{attribute 'linkalways'} 
{attribute 'no_explicit_call' := 'This FB is a CLASS and must be accessed using methods or properties'}
{attribute 'enable_dynamic_creation'}
FUNCTION_BLOCK _TcVnArray7_LREAL EXTENDS AliasDatatypeBase
VAR
	localData : TcVnArray7_LREAL;
	activeData : REFERENCE TO TcVnArray7_LREAL REF= localData;
	aliasBaseDatatype : _Array0to6OfLREAL;
END_VAR

PROPERTY PUBLIC Address : PVOID
GET
Address := ADR(activeData);
END_GET
END_PROPERTY

METHOD PUBLIC ClearReference
VAR_INPUT
END_VAR
activeData REF= localData;
SetBaseDatatypeReference();
END_METHOD

METHOD PUBLIC Clone : I_Datatype
VAR
    pClone : POINTER TO _TcVnArray7_LREAL;
END_VAR
pClone := __NEW(_TcVnArray7_LREAL);
Clone := pClone^;
END_METHOD

METHOD FB_init : BOOL
VAR_INPUT
	bInitRetains : BOOL; // if TRUE, the retain variables are initialized (warm start / cold start)
	bInCopyCode : BOOL;  // if TRUE, the instance afterwards gets moved into the copy code (online change)
	//InitialValue : TcVnArray7_LREAL; // if possible, not all values can be initialized
END_VAR
//localData := InitialValue; // if possible, not all values can be initialized
SetBaseDatatypeReference();
AddBaseDatatype(aliasBaseDatatype);
END_METHOD

PROPERTY PUBLIC Identifier : T_MAXSTRING
GET
Identifier := 'TcVnArray7_LREAL';
END_GET
END_PROPERTY

METHOD PUBLIC MakeReferenceTo
VAR_INPUT
	ReferenceTarget : REFERENCE TO TcVnArray7_LREAL;
END_VAR
activeData REF= ReferenceTarget;
SetBaseDatatypeReference();
END_METHOD

METHOD PROTECTED SetBaseDatatypeReference
VAR_INPUT
END_VAR
aliasBaseDatatype.MakeReferenceTo(activeData);
END_METHOD

PROPERTY PUBLIC Size : UDINT
GET
Size := SIZEOF(activeData);
END_GET
END_PROPERTY

METHOD TryMakeReferenceTo : BOOL
VAR_INPUT
	Target : I_Datatype;
END_VAR
VAR
	pTargetData : POINTER TO TcVnArray7_LREAL;
END_VAR
IF NOT IsEquivalentTo(Target) THEN
	RETURN;
END_IF

pTargetData := Target.Address;
activeData REF= pTargetData^;
SetBaseDatatypeReference();
TryMakeReferenceTo := TRUE;
END_METHOD

PROPERTY PUBLIC Value : REFERENCE TO TcVnArray7_LREAL
GET
Value REF= activeData;
END_GET
END_PROPERTY

END_FUNCTION_BLOCK

(* stored: Version 1.1.0.1, ProductVersion 3.1.4024.13
   POU _TcVnArray7_LREAL: Id {ddf94652-72d9-49c2-8bb5-295fa89ad813}, SpecialFunc None
   Property Address: Id {1fca79c0-d590-4b36-8e8a-9000e6798f50}
   Get Get: Id {a541fe61-ae51-451e-92fa-61de9d520b4d}
   Method ClearReference: Id {27003290-6a62-4b26-a732-a7f67e19df22}
   Method Clone: Id {75c16c64-a72b-4c06-9929-4ae901391bad}
   Method FB_init: Id {5aebf110-a2d0-42f7-817b-a14cd61c5fff}
   Property Identifier: Id {47368d61-7908-48fa-85cb-c11fa4274724}
   Get Get: Id {7f0600d7-46e8-4640-9875-a1adf62abe20}
   Method MakeReferenceTo: Id {18ba65aa-e172-4804-90a5-e60b7482ea29}
   Method SetBaseDatatypeReference: Id {35640ec2-8028-4af7-ae72-a6a1f2831bb6}
   Property Size: Id {89a14830-8edd-4d1b-9f92-593b19920b6a}
   Get Get: Id {b28972ec-7dd7-4cf2-8e7c-b94bc793d5ff}
   Method TryMakeReferenceTo: Id {ca8f5f93-5aa2-4cf6-b1d4-d73d3b41678a}
   Property Value: Id {d2d5116f-1357-4351-be0a-7507ab054c12}
   Get Get: Id {c451c03f-70e5-4e49-97ae-f107899f10a0} *)
